# B&R Automation Studio project kursich
Automation Studio 4.2.10.53 SP

## Configuration Config1

CPU PC_any, AutomationRuntime D4.26, Build 4.1.2, Vc V4.26.5

### Task classes (Cpu.sw)
```
Cyclic#4 (cycle 1000000 us, tolerance 10000000 us):
  Program <- Program.prg
VcDataObjects: Visu <- Visu.dob
Libraries: Library_C
```

### Hardware
```
PC : PC_any v1.1.0.0 (OrderNumber=PC)
  Connector IF3:
    Vnc1
    VncVcObjectName1 = Visu
    VncKeyMappingFile1 = VC\PS2-Keyboard.dis
  ConfigurationID = kursich_Config1
  Cyclic1Duration = 100000
  Cyclic1Tolerance = 10000000
  Cyclic2Duration = 200000
  Cyclic2Tolerance = 10000000
  Cyclic3Duration = 500000
  Cyclic3Tolerance = 10000000
  Cyclic4Duration = 1000000
  Cyclic4Tolerance = 10000000
  Cyclic5Duration = 2000000
  Cyclic5Tolerance = 10000000
  Cyclic6Duration = 3000000
  Cyclic6Tolerance = 12000000
  Cyclic7Duration = 4000000
  Cyclic7Tolerance = 12000000
  Cyclic8Duration = 5000000
  Cyclic8Tolerance = 30000000
  ActivateOpcUa = 1
  OpcUa_Security_SoftwareCertificates = 
```

## Logical view

Binary libraries used (declarations not repeated): operator, runtime, astime, AsIecCon

### Package Logical/Libraries - Global libraries

### Library Logical/Libraries/Library_C (ANSIC)

#### Types.typ - Exported data types
```iecst
TYPE
	ErrorStates :
		(
		NOERROR,
		FALSESTART,
		FALSESTOP,
		FAIL2START,
		FAIL2STOP
		);
	Com_operStates :
		(
		NONE,
		START,
		STOP
		);
	EngineStatusStates :
		(
		STOPPED,
		STARTED,
		TRY2START,
		TRY2STOP
		);
	ValveStatusStates :
		(
		OPENED,
		CLOSED,
		OPENING,
		CLOSING,
		TRY2CLOSE,
		TRY2OPEN
		);
END_TYPE
```

#### Library_C.fun - Exported functions and function blocks
```iecst
FUNCTION_BLOCK Valve
	VAR_INPUT
		ESD_stop : BOOL;
		remote : BOOL := 1;
		local : BOOL;
		CCMCCW : BOOL;
		CCMCW : BOOL;
	END_VAR
	VAR_OUTPUT
		closing : BOOL;
		opening : BOOL;
		open : BOOL;
		ready : BOOL := 1;
		termalTrip : BOOL;
		torqueTrip : BOOL;
		stop : BOOL;
		error : ErrorStates;
	END_VAR
	VAR_IN_OUT
		com_oper : Com_operStates;
	END_VAR
	VAR
		state : ValveStatusStates;
		counter : UINT;
		time2Open : UINT := 10;
		time2Close : UINT := 10;
	END_VAR
END_FUNCTION_BLOCK

FUNCTION_BLOCK Engine (*TODO: Add your comment here*) (*$GROUP=User,$CAT=User,$GROUPICON=User.png,$CATICON=User.png*)
	VAR_INPUT
		ready : BOOL := 1;
		local : BOOL := 0;
		remote : BOOL := 1;
		alarm_stop_button_pressed : BOOL := FALSE;
		time2Start : UINT := 10;
		time2Stop : UINT := 10;
	END_VAR
	VAR_OUTPUT
		error : ErrorStates := NOERROR;
	END_VAR
	VAR_IN_OUT
		com_oper : Com_operStates;
		work : BOOL;
	END_VAR
	VAR
		counter : USINT := 0;
		start : BOOL;
		stop : BOOL;
		state : EngineStatusStates := STOPPED;
	END_VAR
	VAR_OUTPUT
		workTime : UINT;
	END_VAR
END_FUNCTION_BLOCK

FUNCTION_BLOCK Solval
	VAR_INPUT
		ESD_stop : BOOL;
		remote : BOOL := 1;
		local : BOOL;
	END_VAR
	VAR_OUTPUT
		opened : BOOL;
		ready : BOOL := 1;
		openClose : BOOL;
		error : ErrorStates;
	END_VAR
	VAR_IN_OUT
		com_oper : Com_operStates;
	END_VAR
	VAR
		state : ValveStatusStates := CLOSED;
	END_VAR
END_FUNCTION_BLOCK
```

#### Engine.c
```c
#include <bur/plctypes.h>
#ifdef __cplusplus
	extern "C"
	{
#endif
	#include "Library_C.h"
#ifdef __cplusplus
	};
#endif

void Engine(struct Engine* inst)
{
	switch (inst->state) {
		case STOPPED: {
			if(inst->work == 1) {
				inst->state = STARTED;
				break;
			}
			if((inst->com_oper == START) && (inst->ready)) {
				inst->error = NOERROR;
				inst->start = 1;
				inst->work = 1;
				inst->counter = 0;
				inst->com_oper = NONE;
				inst->state = TRY2START;
				break;
			}
		}

		case STARTED: {
			if(inst->work == 0) {
				inst->state = STOPPED;
				break;
			}
			if(inst->com_oper == STOP) {
				inst->error = NOERROR;
				inst->stop = 1;
				inst->work = 0;
				inst->counter = 0;
				inst->com_oper = NONE;
				inst->state = TRY2STOP;
				break;
			}
		}

		case TRY2START: {
			inst->counter += 1;
			if((inst->work == 0) && (inst->counter >= inst->time2Start)) {
				inst->error = FAIL2START;
				inst->start = 0;
				inst->counter = 0;
				inst->state = STOPPED;
				break;
			}
			if(inst->work == 1) {
				inst->start = 1;
				inst->state = STARTED;
				break;
			}
		}

		case TRY2STOP: {
			inst->counter += 1;
			if((inst->work == 1) && (inst->counter >= inst->time2Stop)) {
				inst->error = FAIL2STOP;
				inst->start = 1;
				inst->counter = 0;
				inst->state = STARTED;
				break;
			}
			if(inst->work == 0) {
				inst->start = 0;
				inst->state = STOPPED;
				break;
			}
		}
	}
}
```

#### Valve.c
```c
#include <bur/plctypes.h>
#ifdef __cplusplus
	extern "C"
	{
#endif
	#include "Library_C.h"
#ifdef __cplusplus
	};
#endif
/* TODO: Add your comment here */
void Valve(struct Valve* inst)
{
	switch (inst->state) {
		case CLOSED: {
				if(inst->open == 1) {
					inst->state = OPENED;
					break;
				}
				if((inst->com_oper == START) && (inst->ready)) {
					inst->error = NOERROR;
					inst->counter = 0;
					inst->opening = 1;
					inst->CCMCCW = 1;
					inst->CCMCW = 0;
					inst->stop = 0;
					inst->com_oper = NONE;
					inst->state = TRY2OPEN;
					break;
				}
			}

		case OPENED: {
				if(inst->open == 0) {
					inst->state = CLOSED;
					break;
				}
				if(inst->com_oper == STOP) {
					inst->error = NOERROR;
					inst->counter = 0;
					inst->closing = 1;
					inst->CCMCCW = 0;
					inst->CCMCW = 1;
					inst->stop = 0;
					inst->com_oper = NONE;
					inst->state = TRY2CLOSE;
					break;
				}
			}

		case TRY2OPEN: {
				inst->counter += 1;
				if((inst->opening == 1) && (inst->counter > inst->time2Open)) {
					inst->error = FAIL2START;
					inst->CCMCCW = 0;
					inst->opening = 0;
					inst->stop = 1;
					inst->counter = 0;
					inst->state = CLOSED;
					break;
				}
				if((inst->opening == 1) && (inst->counter = inst->time2Open)) {
					inst->CCMCCW = 0;
					inst->opening = 0;
					inst->open = 1;
					inst->stop = 1;
					inst->state = OPENED;
					break;
				}
			}

		case TRY2CLOSE: {
				inst->counter += 1;
				if((inst->closing == 1) && (inst->counter > inst->time2Close)) {
					inst->error = FAIL2STOP;
					inst->CCMCW = 0;
					inst->closing = 0;
					inst->stop = 1;
					inst->counter = 0;
					inst->state = CLOSED;
					break;
				}
				if((inst->closing == 1) && (inst->counter = inst->time2Close)) {
					inst->CCMCW = 0;
					inst->closing = 0;
					inst->open = 0;
					inst->stop = 1;
					inst->state = CLOSED;
					break;
				}
			}
	}
}
```

#### Solval.c
```c
#include <bur/plctypes.h>
#ifdef __cplusplus
	extern "C"
	{
#endif
	#include "Library_C.h"
#ifdef __cplusplus
	};
#endif
/* TODO: Add your comment here */
void Solval(struct Solval* inst)
{
	switch (inst->state) {
		case CLOSED: {
				if(inst->opened == 1) {
					inst->state = OPENED;
					break;
				}
				if((inst->com_oper == START) && (inst->ready)) {
					inst->error = NOERROR;
					inst->opened = 1;
					inst->com_oper = NONE;
					inst->state = TRY2OPEN;
					break;
				}
			}

		case OPENED: {
				if(inst->opened == 0) {
					inst->state = CLOSED;
					break;
				}
				if(inst->com_oper == STOP) {
					inst->error = NOERROR;
					inst->opened = 0;
					inst->com_oper = NONE;
					inst->state = TRY2CLOSE;
					break;
				}
			}

		case TRY2OPEN: {
				if(inst->opened == 0) {
					inst->error = FAIL2START;
					inst->state = CLOSED;
					break;
				}
				if(inst->opened == 1) {
					inst->state = OPENED;
					break;
				}
			}

		case TRY2CLOSE: {
				if(inst->opened == 1) {
					inst->error = FAIL2STOP;
					inst->state = OPENED;
					break;
				}
				if(inst->opened == 0) {
					inst->state = CLOSED;
					break;
				}
			}
	}
}
```

### Program Logical/Program (ANSIC)

#### Types.typ
```iecst
TYPE
	Com_operStates_G :
		(
		NONE_G,
		START_G,
		STOP_G
		);
END_TYPE
```

#### Variables.var
```iecst
VAR
	CP1 : Engine;
	FAN : Engine;
	DP2 : Engine;
	DP1 : Engine;
	FV1 : Solval;
	MV1 : Valve;
	Level_LL : BOOL;
	Level_L : BOOL;
	RH_LowLimit : INT := 625;
	RH_HighLimit : INT := 630;
	PH_WorkLimit : INT := 8;
	PH_LowLimit : INT := 8;
	Level_H : BOOL;
	Level_HH : BOOL;
	P_HH : BOOL;
	P_LL : BOOL;
	FlowIndic : BOOL;
	RH : INT;
	PH : INT;
	maxWashTimeCP1 : UINT := 10;
	maxFeedTimeDP2 : UINT := 10;
	maxOneTimeFeedDP2 : UINT := 10;
	maxOneTimeFeedDP1 : UINT := 10;
	maxFeedTimeDP1 : UINT := 10;
	TriggersError : BOOL := FALSE;
	com_oper_G : Com_operStates_G := NONE_G;
	visu_L : INT := 252;
	visu_H : INT := 252;
	visu_LL : INT := 252;
	visu_HH : INT := 252;
	visu_CP1 : INT := 252;
	visu_FV1 : INT := 252;
	visu_FAN : INT := 252;
	visu_DP2 : INT := 252;
	visu_DP1 : INT := 252;
	visu_MV1 : INT := 252;
	afterStart : INT := 10;
	ERROR : INT := 252;
END_VAR
```

#### Main.c
```c
#include <bur/plctypes.h>

#ifdef _DEFAULT_INCLUDES
	#include <AsDefault.h>
#endif

void _INIT ProgramInit(void)
{

}

void _CYCLIC ProgramCyclic(void)
{
	Engine(&FAN);
	Engine(&CP1);
	Engine(&DP1);
	Engine(&DP2);
	Solval(&FV1);
	Valve(&MV1);

	if(FAN.work && FlowIndic) {
		if(Level_H && Level_LL && Level_L) {
			if(P_HH == 0) {
				CP1.com_oper = 1;
			}
			if(CP1.work) {
				if(PH <= PH_LowLimit) {
					DP1.com_oper = 1;
				}
				if(RH > RH_HighLimit) {
					DP2.com_oper = 1;
				}
			}
			if((CP1.workTime >= maxWashTimeCP1) || (DP1.workTime >= maxFeedTimeDP1) || (DP2.workTime >= maxFeedTimeDP2)) {
				MV1.com_oper = 1;
			}
		} else {
			if(!(MV1.open)) {
				FV1.com_oper = 1;
			}
		}
	}

	if(!FAN.work || !FlowIndic || !(Level_H && Level_LL && Level_L) || (P_LL && (CP1.workTime > afterStart)) || P_HH) {
		CP1.com_oper = 2;
	}
	if(!FAN.work || !FlowIndic || !(Level_H && Level_LL && Level_L) || !(CP1.work) || (PH > PH_WorkLimit) || (DP1.workTime >= maxOneTimeFeedDP1)) {
		DP1.com_oper = 2;
	}
	if(!FAN.work || !FlowIndic || !(Level_H && Level_LL && Level_L) || !(CP1.work) || (RH < RH_LowLimit) || (DP2.workTime >= maxOneTimeFeedDP2)) {
		DP2.com_oper = 2;
	}
	if(!FAN.work || !FlowIndic || (Level_H && Level_LL && Level_L) || MV1.open) {
		FV1.com_oper = 2;
	}
	if(!FAN.work || !FlowIndic || !(Level_H && Level_LL && Level_L)) {
		MV1.com_oper = 2;
	}

	if(Level_HH || (Level_H && ((!(Level_L) || !(Level_LL)))) || (!(Level_H) && !(Level_LL) && Level_L)) {
		TriggersError = 1;
		FAN.com_oper = 2;
		CP1.com_oper = 2;
		DP1.com_oper = 2;
		DP2.com_oper = 2;
		FV1.com_oper = 2;
		MV1.com_oper = 2;
	} else {
		TriggersError = 0;
	}
	if(TriggersError) {
		if(ERROR == 0) {
			ERROR = 51;
		} else {
			ERROR = 0;
		}
	} else {
		ERROR = 252;
	}

	if(Level_LL) {
		visu_LL = 11;
	} else {
		visu_LL = 252;
	}
	if(Level_L) {
		visu_L = 11;
	} else {
		visu_L = 252;
	}
	if(Level_H) {
		visu_H = 11;
	} else {
		visu_H = 252;
	}
	if(Level_HH) {
		visu_HH = 11;
	} else {
		visu_HH = 252;
	}

	if(FAN.work) {
		visu_FAN = 226;
	} else {
		visu_FAN = 252;
	}
	if(CP1.work) {
		visu_CP1 = 226;
	} else {
		visu_CP1 = 252;
	}
	if(FV1.opened) {
		visu_FV1 = 226;
	} else {
		visu_FV1 = 252;
	}
	if(MV1.open) {
		visu_MV1 = 226;
	} else {
		visu_MV1 = 252;
	}
	if(DP1.work) {
		visu_DP1 = 226;
	} else {
		visu_DP1 = 252;
	}
	if(DP2.work) {
		visu_DP2 = 226;
	} else {
		visu_DP2 = 252;
	}
}
void _EXIT ProgramExit(void)
{
	// Insert code here

}
```

- Visualisation Logical/Visu (not shown)

Listed in the project but not available here: Logical/Global.typ, Logical/Global.var, Logical/Libraries/Library_C/Constants.var
